FUNCTION_BLOCK FB_HMI_TP_BRANCH_A EXTENDS FB_HMI_COMPONENT
VAR_INPUT
END_VAR
VAR_OUTPUT
END_VAR
VAR
END_VAR

END_FUNCTION_BLOCK

(* stored: Version 1.1.0.1, ProductVersion 3.1.4024.14
   POU FB_HMI_TP_BRANCH_A: Id {eae4b508-ce15-49d6-ac96-db77702b1c9c}, SpecialFunc None *)
